TEXTLIST textListRight
  0 = ''
  1 = 'X'
  2 = '>'
  3 = '<'
   = ''
END_TEXTLIST

(* stored: Version 1.1.0.1, ProductVersion 3.1.4024.11
   TextList textListRight: Id {04ce01a3-180f-03be-0fae-0aa9cfb08bb5} *)
